RoboDK station: AROB_S4_A5.rdk

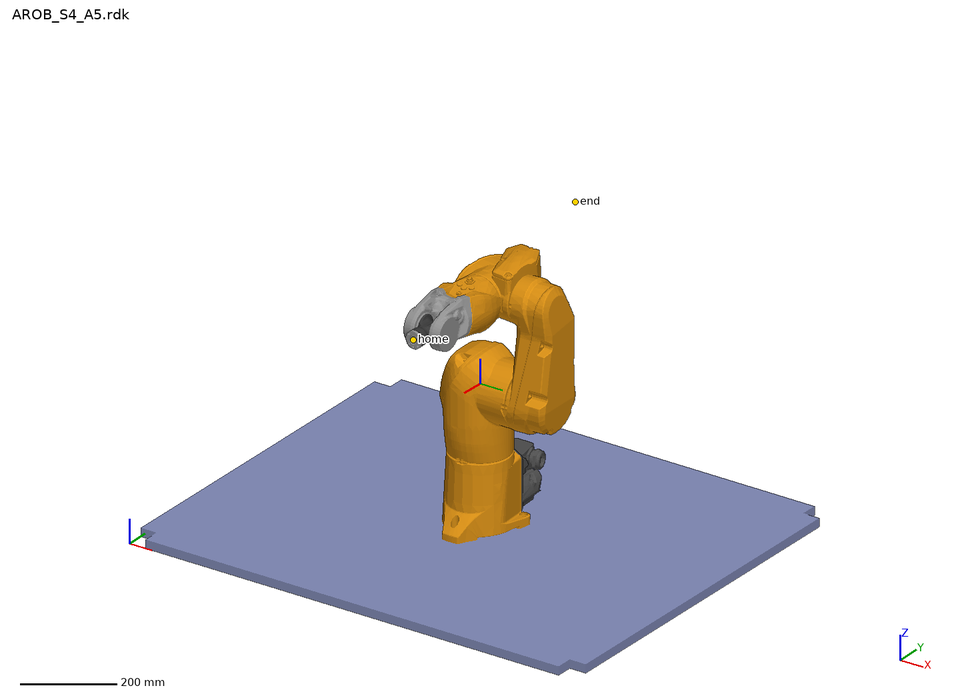
[picture v0: the station drawn from its stored meshes, robots at their saved joint values, targets as dots, program paths as lines]
Station AROB_S4_A5 (saved by RoboDK 5.6.9). Poses are relative to the parent item; angles as X-Y-Z fixed-axis rotations.
  - frame world at (0, 0, 0) mm
    - frame Staubli TX2-40 Base at (560, 460, 340) mm, rotated rx 0 ry 0 rz -90 deg
      - robot Staubli TX2-40: 6 axes, payload 2 kg, reach 515 mm, repeatability 0.02 mm, weight 29 kg
          modified DH rows (alpha deg, a mm, theta deg, d mm): 0, 0, 0, 320; -90, 0, -90, 35; 0, 225, -90, 0; -90, 0, 0, 225; 90, 0, 0, 0; -90, 0, 180, 65
          base shift (0, 0, -320) mm
          joint limits [-180, -125, -138, -270, -120, -270] to [180, 125, 138, 270, 133.5, 270]; home [0, 0, 90, 0, 0, 0]; saved at [0, 0, 90, 0, 0, 0]
    - object Arbeitsflaeche_geteilt at (0, 0, 0) mm, size 1120 x 920 x 20 mm, geometry from Arbeitsflaeche_geteilt.iges
    - object Arbeitsflaeche_komplett at (0, 0, 0) mm, size 1120 x 920 x 20 mm, geometry from Arbeitsflaeche_komplett.IGS
    - object Zelle at (0, 0, 0) mm, rotated rx 90 ry 0 rz -90 deg, size 1120 x 1947.8 x 1200 mm, geometry from Zelle.stp
    - target home (joint target) at (595, 170, 565) mm, rotated rx 0 ry 90 rz -90 deg; joints [0, 0, 90, 0, 0, 0] of Staubli TX2-40
    - target end (joint target) at (730.33, 559.49, 764.49) mm, rotated rx 62.55 ry 25.09 rz 78.25 deg; joints [118, 0, 40, -50, 33, 95] of Staubli TX2-40
    - target Target 1 (joint target) at (595, 170, 565) mm, rotated rx 0 ry 90 rz -90 deg; joints [39.333, 0, 73.333, -16.667, 11, 31.667] of Staubli TX2-40
    - target Target 2 (joint target) at (595, 170, 565) mm, rotated rx 0 ry 90 rz -90 deg; joints [78.667, 0, 56.667, -33.333, 22, 63.333] of Staubli TX2-40
  - Python program Prog_viaTarget (listed below)
  - Python program Prog_Direct (listed below)
  - Python program Prog_Collision (listed below)

--- Python program Prog_viaTarget ---
# Type help("robodk.robolink") or help("robodk.robomath") for more information
# Press F5 to run the script
# Documentation: https://robodk.com/doc/en/RoboDK-API.html
# Reference:     https://robodk.com/doc/en/PythonAPI/robodk.html
# Note: It is not required to keep a copy of this file, your Python script is saved with your RDK project
import robodk.robolink as rl    # Robot link toolbox
import time

# Link to RoboDK
RDK = rl.Robolink()

robot = RDK.Item('Staubli TX2-40')
world = RDK.Item('world')


n = 10


target1 = RDK.Item('Target 1')

target2 = RDK.Item('Target 2')
target3 = RDK.Item('Target 3')
target4 = RDK.Item('Target 4')
target5 = RDK.Item('Target 5')
end = RDK.Item('end')

print('start')

robot.setAccelerationJoints(150)
robot.setSpeedJoints(75)

robot.MoveJ(home)
robot.MoveJ(target1)
robot.MoveJ(target2)
robot.MoveJ(target3)
robot.MoveJ(target4)
robot.MoveJ(target5)
robot.MoveJ(end)
time.sleep(0.1)
robot.MoveJ(target5)
robot.MoveJ(target4)
robot.MoveJ(target3)
robot.MoveJ(target2)
robot.MoveJ(target1)
robot.MoveJ(home)
print('end')

--- Python program Prog_Direct ---
# Type help("robodk.robolink") or help("robodk.robomath") for more information
# Press F5 to run the script
# Documentation: https://robodk.com/doc/en/RoboDK-API.html
# Reference:     https://robodk.com/doc/en/PythonAPI/robodk.html
# Note: It is not required to keep a copy of this file, your Python script is saved with your RDK project
import robodk.robolink as rl    # Robot link toolbox
import time
import numpy as np

# Link to RoboDK
RDK = rl.Robolink()

robot = RDK.Item('Staubli TX2-40')
world = RDK.Item('world')
home = RDK.Item('home')
target1 = RDK.Item('Target 1')
target2 = RDK.Item('Target 2')
target3 = RDK.Item('Target 3')
target4 = RDK.Item('Target 4')
target5 = RDK.Item('Target 5')
end = RDK.Item('end')

print(target1)

print('start')

robot.setAccelerationJoints(150)
robot.setSpeedJoints(75)

robot.MoveJ(home)
robot.MoveJ(end)

time.sleep(0.1)

robot.MoveJ(home)
print('end')

--- Python program Prog_Collision ---
# Type help("robodk.robolink") or help("robodk.robomath") for more information
# Press F5 to run the script
# Documentation: https://robodk.com/doc/en/RoboDK-API.html
# Reference:     https://robodk.com/doc/en/PythonAPI/robodk.html
# Note: It is not required to keep a copy of this file, your Python script is saved with your RDK project

# You can also use the new version of the API:
import robodk.robolink as rl    # RoboDK API
import robodk.robomath as rm    # Robot toolbox
import numpy as np
RDK = rl.Robolink()

target_list_names = RDK.ItemList(filter=rl.ITEM_TYPE_TARGET,list_names=True)

for target_name in target_list_names:
    if 'Target' in target_name:
        print(target_name)
        RDK.Delete(RDK.Item(target_name))


home= RDK.Item('home')
robot = RDK.Item('Staubli TX2-40')
world = RDK.Item('world')
end = RDK.Item('end')

theta_i = np.array([   0.0, -90.0,  90.0,   0.0,   0.0,   0.0])
d_i =     np.array([   0.0,  35.0,   0.0, 225.0,   0.0,  65.0])
a_i =     np.array([   0.0, 225.0,   0.0,   0.0,   0.0,   0.0])
alpha_i = np.array([ -90.0,   0.0,  90.0, -90.0,  90.0,   0.0])



theta_start = np.array([   0.0,  0.0, 90.0,   0.0,  0.0,  0.0])
theta_end   = np.array([ 118.0,  0.0, 40.0, -50.0, 33.0, 95.0])
theta_midpoints = np.array([0,0,0,0,0,0])
n_midpoints = 2

theta_difference = theta_end - theta_start
theta_steps = theta_difference/(n_midpoints + 1)

targets = [None] * n_midpoints

for i in range(0, n_midpoints):
    targets[i] = RDK.AddTarget('Target ' + str(i + 1), world).setAsJointTarget()
    theta = theta_steps * (i + 1) + theta_start
    targets[i].setJoints([theta[0],theta[1],theta[2],theta[3],theta[4],theta[5]])

print('start')

robot.setAccelerationJoints(10)
robot.setSpeedJoints(10)

robot.MoveJ(home)

for i in range(0, n_midpoints):
    robot.MoveJ(targets[i])

robot.MoveJ(end)

for i in range(n_midpoints-1, -1, -1):
    robot.MoveJ(targets[i])

robot.MoveJ(home)
